// TIA Portal V17 export
// export: Created 2025-03-05T08:03:42.7657928Z, ExportSetting WithDefaults, DisplayName Totally Integrated Automation Portal, DisplayVersion V17 Update 8, DisplayName TIA Portal Openness, DisplayVersion V17 Update 8, DisplayName TIA Portal Version Control Interface, DisplayVersion V17, DisplayName SINAMICS Startdrive Advanced, DisplayVersion V17 SP2, DisplayName SINAMICS Startdrive G110M, G120, G120C, G120D, G120P, G115D, DisplayVersion V17 SP2, DisplayName SINAMICS Startdrive G130, G150, S120, S150, SINAMICS MV, S210, DisplayVersion V17 SP2, DisplayName STEP 7 Professional, DisplayVersion V17 Update 8, DisplayName SINUMERIK ONE STEP 7 Toolbox, DisplayVersion V17 Update 12, DisplayName SINUMERIK 840D sl STEP 7 Toolbox, DisplayVersion V17 Update 12, DisplayName STEP 7 Safety, DisplayVersion V17 Update 6, DisplayName WinCC Advanced, DisplayVersion V17 Update 8
TYPE "GENERAL_DATA_SEQUENCES"
// stored: IsFailsafeCompliant false
   STRUCT
      START_GENERAL_CONDITIONS : Bool;   // Start general conditions
      START_GENERAL_CONDITIONS_HELP : Bool;   // Start general conditions help
      START_INITIAL_CONDITIONS : Bool;   // Start initial conditions
      START_INITIAL_CONDITIONS_HELP : Bool;   // Start initial conditions help
      START_MANUAL_REQUEST : Bool;   // Start manual request
      START_SEMI_REQUEST : Bool;   // Start semi request
      START_AUTO_REQUEST : Bool;   // Start auto request
      START_COMMAND : Bool;   // Start command
      STOP_GENERAL_CONDITIONS : Bool;   // Stop general conditions
      STOP_GENERAL_CONDITIONS_HELP : Bool;   // Stop general conditions help
      STOP_INITIAL_CONDITIONS : Bool;   // Stop initial conditions
      STOP_INITIAL_CONDITIONS_HELP : Bool;   // Stop initial conditions help
      STOP_MANUAL_CONDITIONS : Bool;   // Stop manual conditions
      STOP_MANUAL_REQUEST : Bool;   // Stop manual request
      STOP_SEMI_REQUEST : Bool;   // Stop semi request
      STOP_AUTO_REQUEST : Bool;   // Stop auto request
      STOP_COMMAND : Bool;   // Stop command
      SEQUENCE_RUNNING : Bool;   // Sequence running
      STEP_1 : Bool;   // Step 1
      STEP_2 : Bool;   // Step 2
      STEP_3 : Bool;   // Step 3
      STEP_4 : Bool;   // Step 4
      STEP_5 : Bool;   // Step 5
      STEP_6 : Bool;   // Step 6
      STEP_7 : Bool;   // Step 7
      STEP_8 : Bool;   // Step 8
      STEP_9 : Bool;   // Step 9
      STEP_10 : Bool;   // Step 10
      STEP_11 : Bool;   // Step 11
      STEP_12 : Bool;   // Step 12
      RESET_PLC_SEQUENCE : Bool;   // Reset PLC sequence
      SEQUENCE_DONE : Bool;   // Sequence done
      SEQUENCE_EXCEEDED_TIME : Bool;   // Sequence exceeded time
      WARNING : Bool;   // Warning
   END_STRUCT;
END_TYPE
